TEXTLIST coloresSensorVision
  3 = 'Azul'
  6 = 'Verde'
  9 = 'Metal'
  0 = '-'
   = ''
END_TEXTLIST

(* stored: Version 1.1.0.1, ProductVersion 3.1.4024.15
   TextList coloresSensorVision: Id {a0d3362d-c2af-406c-9471-d60cefda2e40} *)
